// TIA Portal V19 export
FUNCTION "FC_Anf_BE" : Void   // FC31, LAD
TITLE = Anforderung WR02 /WR03 in Automatik
{ S7_Optimized_Access := 'TRUE' }
// stored: AutoNumber false, SetENOAutomatically false
   VAR_INPUT
      Req_GO_Ausfahrt : Bool;
      Req_GO_Aufgabe : Bool;
   END_VAR
   VAR_IN_OUT
      Req_WR02_IN : Bool;
      Req_WR02_OUT : Bool;
      Req_WR03_IN : Bool;
      Req_WR03_OUT : Bool;
   END_VAR
   VAR_TEMP
      alles_frei : Bool;
      Korb_in_Anlage : Bool;
      BE1_inA : Bool;
      BE1_outA : Bool;
      BE2_inA : Bool;
      BE2_outA : Bool;
      BE3_inA : Bool;
      BE3_outA : Bool;
      BE4_inA : Bool;
      BE4_outA : Bool;
      BE5_inA : Bool;
      BE5_outA : Bool;
      BE6_inA : Bool;
      BE6_outA : Bool;
      links_ok : Bool;
      rechts_ok : Bool;
      WT_DB_Nr : Word;
   END_VAR
BEGIN

REGION Network 1 (SCL): Check Zustand
   // Hat was zu tun
   IF (#Req_WR02_IN OR #Req_WR02_OUT) OR (#Req_WR03_IN OR #Req_WR03_OUT) THEN
       RETURN;
   END_IF;
   // TW hat Befehl
   IF "DB_POS".POS[25].Quelle OR "DB_POS".POS[25].Ziel OR "DB_POS".POS[26].Quelle OR "DB_POS".POS[26].Ziel OR
       "DB_POS".POS[27].Quelle OR "DB_POS".POS[27].Ziel OR "DB_POS".POS[28].Quelle OR "DB_POS".POS[28].Ziel OR
       "DB_POS".POS[29].Quelle OR "DB_POS".POS[29].Ziel OR "DB_POS".POS[30].Quelle OR "DB_POS".POS[30].Ziel THEN
       RETURN;
   END_IF;

   // Kompleett leer
   #alles_frei := NOT "DB_BE_Stand".Stand[1].IN_Belegt AND NOT "DB_BE_Stand".Stand[2].IN_Belegt AND
   NOT "DB_BE_Stand".Stand[3].IN_Belegt AND NOT "DB_BE_Stand".Stand[4].IN_Belegt AND
   NOT "DB_BE_Stand".Stand[5].IN_Belegt AND NOT "DB_BE_Stand".Stand[6].IN_Belegt;
   // mindestens 1 Korb in der Anlage
   #Korb_in_Anlage := ("DB_POS".POS[1].next_WT + "DB_POS".POS[2].next_WT + "DB_POS".POS[3].next_WT + "DB_POS".POS[4].next_WT + "DB_POS".POS[5].next_WT + "DB_POS".POS[6].next_WT
       + "DB_POS".POS[7].next_WT + "DB_POS".POS[8].next_WT + "DB_POS".POS[9].next_WT + "DB_POS".POS[10].next_WT + "DB_POS".POS[11].next_WT + "DB_POS".POS[12].next_WT
       + "DB_POS".POS[13].next_WT + "DB_POS".POS[14].next_WT + "DB_POS".POS[15].next_WT + "DB_POS".POS[16].next_WT +"DB_POS".POS[17].next_WT + "DB_POS".POS[18].next_WT
       + "DB_POS".POS[19].next_WT + "DB_POS".POS[20].next_WT + "DB_POS".POS[21].next_WT + "DB_POS".POS[22].next_WT +"DB_POS".POS[23].next_WT + "DB_POS".POS[24].next_WT
       ) > 0;
END_REGION

NETWORK
TITLE = in die Anlage / aus der Anlage ?
      L     0;
      L     "DB_POS".POS[25].WT_DB;
      >=I;
      R     #BE1_inA;
      R     #BE1_outA;
      JC    BE_2;
      L     "DB_POS".POS[25].WT_DB;
      +     +100;
      T     #WT_DB_Nr;
      OPN   DB [#WT_DB_Nr];
      A     %DBX18.1;  //"DB_WTx".in_Anlage
      S     #BE1_inA;
      R     #BE1_outA;
      JC    BE_2;
      A     %DBX18.3;  //"DB_WTx".aus_Anlage
      S     #BE1_outA;
      R     #BE1_inA;

BE_2: L     0;
      L     "DB_POS".POS[26].WT_DB;
      >=I;
      R     #BE2_inA;
      R     #BE2_outA;
      JC    BE_3;
      L     "DB_POS".POS[26].WT_DB;
      +     +100;
      T     #WT_DB_Nr;
      OPN   DB [#WT_DB_Nr];
      A     %DBX18.1;  //"DB_WTx".in_Anlage
      S     #BE2_inA;
      R     #BE2_outA;
      JC    BE_3;
      A     %DBX18.3;  //"DB_WTx".aus_Anlage
      S     #BE2_outA;
      R     #BE2_inA;

BE_3: L     0;
      L     "DB_POS".POS[27].WT_DB;
      >=I;
      R     #BE3_inA;
      R     #BE3_outA;
      JC    BE_4;
      L     "DB_POS".POS[27].WT_DB;
      +     +100;
      T     #WT_DB_Nr;
      OPN   DB [#WT_DB_Nr];
      A     %DBX18.1;  //"DB_WTx".in_Anlage
      S     #BE3_inA;
      R     #BE3_outA;
      JC    BE_4;
      A     %DBX18.3;  //"DB_WTx".aus_Anlage
      S     #BE3_outA;
      R     #BE3_inA;

BE_4: L     0;
      L     "DB_POS".POS[28].WT_DB;
      >=I;
      R     #BE4_inA;
      R     #BE4_outA;
      JC    BE_5;
      L     "DB_POS".POS[28].WT_DB;
      +     +100;
      T     #WT_DB_Nr;
      OPN   DB [#WT_DB_Nr];
      A     %DBX18.1;  //"DB_WTx".in_Anlage
      S     #BE4_inA;
      R     #BE4_outA;
      JC    BE_5;
      A     %DBX18.3;  //"DB_WTx".aus_Anlage
      S     #BE4_outA;
      R     #BE4_inA;

BE_5: L     0;
      L     "DB_POS".POS[29].WT_DB;
      >=I;
      R     #BE5_inA;
      R     #BE5_outA;
      JC    BE_6;
      L     "DB_POS".POS[29].WT_DB;
      +     +100;
      T     #WT_DB_Nr;
      OPN   DB [#WT_DB_Nr];
      A     %DBX18.1;  //"DB_WTx".in_Anlage
      S     #BE5_inA;
      R     #BE5_outA;
      JC    BE_6;
      A     %DBX18.3;  //"DB_WTx".aus_Anlage
      S     #BE5_outA;
      R     #BE5_inA;

BE_6: L     0;
      L     "DB_POS".POS[30].WT_DB;
      >=I;
      R     #BE6_inA;
      R     #BE6_outA;
      JC    BE_E;
      L     "DB_POS".POS[30].WT_DB;
      +     +100;
      T     #WT_DB_Nr;
      OPN   DB [#WT_DB_Nr];
      A     %DBX18.1;  //"DB_WTx".in_Anlage
      S     #BE6_inA;
      R     #BE6_outA;
      JC    BE_E;
      A     %DBX18.3;  //"DB_WTx".aus_Anlage
      S     #BE6_outA;
      R     #BE6_inA;

BE_E: NOP   0;


REGION Network 3 (SCL): Großoptik
   IF #Req_GO_Ausfahrt  OR #BE3_outA  OR #BE4_outA THEN
       // Warten auf Korb
       IF "DB_BE_Stand".Stand[3].IN_innen AND #alles_frei THEN
           RETURN;
       END_IF;
       // Fertigware Raus
       #links_ok := #BE3_outA AND NOT #BE4_inA AND NOT #BE2_inA AND NOT #BE6_inA;

       #rechts_ok := #BE4_outA AND NOT #BE3_inA AND NOT #BE1_inA AND NOT #BE5_inA;

       IF "DB_BE_Stand".Stand[3].IN_innen AND (#links_ok OR #rechts_ok) THEN
           #Req_WR02_OUT := #Req_WR03_OUT :=TRUE;
           RETURN;
       END_IF;
       // Leer Rein
       IF NOT "DB_BE_Stand".Stand[3].IN_innen AND #alles_frei THEN
           #Req_WR02_IN := #Req_WR03_IN := TRUE;
           RETURN;
       END_IF;
    END_IF;

    IF #Req_GO_Aufgabe OR #BE3_inA  OR #BE4_inA  THEN
        // Warten auf Korb
        IF "DB_BE_Stand".Stand[3].IN_aussen AND #alles_frei THEN
            RETURN;
        END_IF;
        // Rohware --> Rein BE3 / BE4
        #links_ok := #BE3_inA AND "DB_BE_Stand".Stand[3].IN_Freigabe AND NOT #BE4_outA
        AND (#BE2_inA AND  "DB_BE_Stand".Stand[2].IN_Freigabe OR NOT "DB_BE_Stand".Stand[2].IN_Belegt)
        AND (#BE6_inA AND  "DB_BE_Stand".Stand[6].IN_Freigabe OR NOT "DB_BE_Stand".Stand[6].IN_Belegt);

        #rechts_ok := #BE4_inA AND "DB_BE_Stand".Stand[4].IN_Freigabe AND NOT #BE3_outA
        AND (#BE1_inA AND  "DB_BE_Stand".Stand[1].IN_Freigabe OR NOT "DB_BE_Stand".Stand[1].IN_Belegt)
        AND (#BE5_inA AND  "DB_BE_Stand".Stand[5].IN_Freigabe OR NOT "DB_BE_Stand".Stand[5].IN_Belegt);

        IF "DB_BE_Stand".Stand[3].IN_aussen AND (#links_ok OR #rechts_ok) THEN
            #Req_WR02_IN := #Req_WR03_IN := TRUE;
            RETURN;
        END_IF;
        // Leer Raus
        IF NOT "DB_BE_Stand".Stand[3].IN_aussen AND #alles_frei THEN
            #Req_WR02_OUT := #Req_WR03_OUT := TRUE;
            RETURN;
        END_IF;
    END_IF;
END_REGION

REGION Network 4 (SCL): Schmalware (kurz oder lang)
   // Warten auf Korb
   IF #alles_frei AND (("DB_BE_Stand".Stand[1].IN_aussen AND "DB_BE_Stand".Stand[5].IN_innen) OR ("DB_BE_Stand".Stand[5].IN_aussen AND "DB_BE_Stand".Stand[1].IN_innen)) THEN
       RETURN;
   END_IF;

   // Fertigware Raus BE1
   IF "DB_BE_Stand".Stand[1].IN_innen AND ((#BE1_outA AND NOT #BE2_inA) OR (#BE2_outA AND NOT #BE1_inA)) THEN
       #Req_WR02_OUT := TRUE;
       IF "DB_BE_Stand".Stand[5].IN_aussen AND NOT "DB_BE_Stand".Stand[5].IN_Belegt AND NOT "DB_BE_Stand".Stand[6].IN_Belegt AND #Korb_in_Anlage THEN
           #Req_WR03_IN := TRUE;
       END_IF;
       RETURN;
   END_IF;
   // Fertigware Raus BE5
   IF "DB_BE_Stand".Stand[5].IN_innen AND ((#BE5_outA AND NOT #BE6_inA) OR (#BE6_outA AND NOT #BE5_inA)) THEN
       #Req_WR03_OUT := TRUE;
       IF "DB_BE_Stand".Stand[1].IN_aussen AND NOT "DB_BE_Stand".Stand[1].IN_Belegt AND NOT "DB_BE_Stand".Stand[2].IN_Belegt AND #Korb_in_Anlage THEN
           #Req_WR02_IN := TRUE;
       END_IF;
       RETURN;
   END_IF;
   // Rohware --> Rein BE1 / BE2
   IF "DB_BE_Stand".Stand[1].IN_aussen AND ((#BE1_inA AND "DB_BE_Stand".Stand[1].IN_Freigabe AND NOT #BE2_outA) OR (#BE2_inA AND "DB_BE_Stand".Stand[2].IN_Freigabe AND NOT #BE1_outA)) THEN
       #Req_WR02_IN := TRUE;
       IF "DB_BE_Stand".Stand[5].IN_innen AND NOT "DB_BE_Stand".Stand[5].IN_Belegt AND NOT "DB_BE_Stand".Stand[6].IN_Belegt THEN
           #Req_WR03_OUT := TRUE;
       END_IF;
       RETURN;
   END_IF;
   // Rohware --> Rein BE5 / BE6
   IF "DB_BE_Stand".Stand[5].IN_aussen AND ((#BE5_inA AND "DB_BE_Stand".Stand[5].IN_Freigabe AND NOT #BE6_outA) OR (#BE6_inA AND "DB_BE_Stand".Stand[6].IN_Freigabe AND  NOT #BE5_outA)) THEN
       #Req_WR03_IN := TRUE;
       IF "DB_BE_Stand".Stand[1].IN_innen AND NOT "DB_BE_Stand".Stand[1].IN_Belegt AND NOT "DB_BE_Stand".Stand[2].IN_Belegt THEN
           #Req_WR02_OUT := TRUE;
       END_IF;
       RETURN;
   END_IF;

   // Beide drin 
   IF "DB_BE_Stand".Stand[1].IN_innen AND "DB_BE_Stand".Stand[5].IN_innen THEN
       IF NOT "DB_BE_Stand".Stand[1].IN_Belegt AND NOT "DB_BE_Stand".Stand[2].IN_Belegt AND NOT "DB_BE_Stand".Stand[3].IN_Belegt AND NOT "DB_BE_Stand".Stand[4].IN_Belegt THEN
           #Req_WR02_OUT := TRUE;
           RETURN;
       END_IF;
       IF NOT "DB_BE_Stand".Stand[5].IN_Belegt AND NOT "DB_BE_Stand".Stand[6].IN_Belegt AND NOT "DB_BE_Stand".Stand[3].IN_Belegt AND NOT "DB_BE_Stand".Stand[4].IN_Belegt THEN
           #Req_WR03_OUT := TRUE;
           RETURN;
       END_IF;
   END_IF;

   // Beide draussen und min. 1 Korb in Anlage
   IF "E_T_Frg_BE" AND "DB_BE_Stand".Stand[1].IN_aussen AND "DB_BE_Stand".Stand[5].IN_aussen AND #Korb_in_Anlage THEN
       IF NOT "DB_BE_Stand".Stand[1].IN_Belegt AND NOT "DB_BE_Stand".Stand[2].IN_Belegt AND NOT "DB_BE_Stand".Stand[3].IN_Belegt AND NOT "DB_BE_Stand".Stand[4].IN_Belegt THEN
           #Req_WR02_IN := TRUE;
           RETURN;
       END_IF;
       IF NOT "DB_BE_Stand".Stand[5].IN_Belegt AND NOT "DB_BE_Stand".Stand[6].IN_Belegt AND NOT "DB_BE_Stand".Stand[3].IN_Belegt AND NOT "DB_BE_Stand".Stand[4].IN_Belegt THEN
           #Req_WR03_IN := TRUE;
           RETURN;
       END_IF;
   END_IF;
END_REGION
END_FUNCTION
